Universal Robots PolyScope program: eris_v2.urp

Program eris_v2 (installation=repl_installation directory=/programs createdIn=5.16.0 lastSavedIn=5.16.0 robotSerialNumber=20185501065)
Calibrated DH parameters: a=[0.000073, -0.261994, -0.164879, -0.000046, 0.000172, 0]; d=[0.162442, 111.219294, -268.471343, 157.385991, 0.099874, 0.099634]; alpha=[1.569873, -0.003012, -0.002263, 1.572206, -1.569596, 0]; deltaTheta=[0, -0.907061, 8.327173, -1.13692, -0.000001, 0]
InitVariablesNode
Robot Program (runOnlyOnce=false)
  Script file /programs/script_code.script
    | socket_open("192.168.1.15", 8000, "abcd")
    | 
    | a = p[-0.421, -0.436, 0.1, 2.61, -1.806, -0.019]
    | # movej(a, a=0.3, v=0.3)
    | 
    | b = p[-0.194, -0.6, 0.066, 2.61, -1.806, -0.019]
    | 
    | i = 0
    | while i < 5:
    |     sleep(2)
    |     i = i + 1
    | end
    | 
    | # movej(b, a=0.3, v=0.3)
